GLOBALCONSTANTS DefaultPool_PI_Numeric (* Numeric object pool constants (ID, Scale, Offset, Decimals) *)
  PACKAGE Uebungen::const::UT::PI;
  VAR_GLOBAL CONSTANT
    OutputNumber_c1_N : logiBUS::utils::conversion::phys::NumericObjectPool_S := (u16ObjId := 12001, r32Scale := 1.0, i32Offset := 0, u8Decimals := 0);
    OutputNumber_c9_N : logiBUS::utils::conversion::phys::NumericObjectPool_S := (u16ObjId := 12009, r32Scale := 1.0, i32Offset := 0, u8Decimals := 0);
    OutputNumber_c10_N : logiBUS::utils::conversion::phys::NumericObjectPool_S := (u16ObjId := 12010, r32Scale := 1.0, i32Offset := 0, u8Decimals := 0);
    OutputNumber_c11_N : logiBUS::utils::conversion::phys::NumericObjectPool_S := (u16ObjId := 12011, r32Scale := 1.0, i32Offset := 0, u8Decimals := 0);
    OutputNumber_c12_N : logiBUS::utils::conversion::phys::NumericObjectPool_S := (u16ObjId := 12012, r32Scale := 1.0, i32Offset := 0, u8Decimals := 0);
    OutputNumber_c2_N : logiBUS::utils::conversion::phys::NumericObjectPool_S := (u16ObjId := 12013, r32Scale := 1.0, i32Offset := 0, u8Decimals := 0);
    OutputNumber_c3_N : logiBUS::utils::conversion::phys::NumericObjectPool_S := (u16ObjId := 12014, r32Scale := 1.0, i32Offset := 0, u8Decimals := 0);
    OutputNumber_c4_N : logiBUS::utils::conversion::phys::NumericObjectPool_S := (u16ObjId := 12015, r32Scale := 1.0, i32Offset := 0, u8Decimals := 0);
    OutputNumber_c5_N : logiBUS::utils::conversion::phys::NumericObjectPool_S := (u16ObjId := 12016, r32Scale := 1.0, i32Offset := 0, u8Decimals := 0);
    OutputNumber_c6_N : logiBUS::utils::conversion::phys::NumericObjectPool_S := (u16ObjId := 12017, r32Scale := 1.0, i32Offset := 0, u8Decimals := 0);
    OutputNumber_c7_N : logiBUS::utils::conversion::phys::NumericObjectPool_S := (u16ObjId := 12018, r32Scale := 1.0, i32Offset := 0, u8Decimals := 0);
    OutputNumber_c8_N : logiBUS::utils::conversion::phys::NumericObjectPool_S := (u16ObjId := 12019, r32Scale := 1.0, i32Offset := 0, u8Decimals := 0);
    OutputNumber_Tick_N : logiBUS::utils::conversion::phys::NumericObjectPool_S := (u16ObjId := 12020, r32Scale := 1.0, i32Offset := 0, u8Decimals := 0);
    OutputNumber_PI_I01_FREQ_N : logiBUS::utils::conversion::phys::NumericObjectPool_S := (u16ObjId := 12021, r32Scale := 1.0, i32Offset := 0, u8Decimals := 0);
    OutputNumber_PI_I01_COUNT_N : logiBUS::utils::conversion::phys::NumericObjectPool_S := (u16ObjId := 12022, r32Scale := 1.0, i32Offset := 0, u8Decimals := 0);
    OutputNumber_PI_I02_FREQ_N : logiBUS::utils::conversion::phys::NumericObjectPool_S := (u16ObjId := 12023, r32Scale := 1.0, i32Offset := 0, u8Decimals := 0);
    OutputNumber_PI_I02_COUNT_N : logiBUS::utils::conversion::phys::NumericObjectPool_S := (u16ObjId := 12024, r32Scale := 1.0, i32Offset := 0, u8Decimals := 0);
    OutputNumber_PI_I03_FREQ_N : logiBUS::utils::conversion::phys::NumericObjectPool_S := (u16ObjId := 12025, r32Scale := 1.0, i32Offset := 0, u8Decimals := 0);
    OutputNumber_PI_I03_COUNT_N : logiBUS::utils::conversion::phys::NumericObjectPool_S := (u16ObjId := 12026, r32Scale := 1.0, i32Offset := 0, u8Decimals := 0);
    OutputNumber_PI_I04_FREQ_N : logiBUS::utils::conversion::phys::NumericObjectPool_S := (u16ObjId := 12027, r32Scale := 1.0, i32Offset := 0, u8Decimals := 0);
    OutputNumber_PI_I04_COUNT_N : logiBUS::utils::conversion::phys::NumericObjectPool_S := (u16ObjId := 12028, r32Scale := 1.0, i32Offset := 0, u8Decimals := 0);
    OutputNumber_PI_I05_FREQ_N : logiBUS::utils::conversion::phys::NumericObjectPool_S := (u16ObjId := 12029, r32Scale := 1.0, i32Offset := 0, u8Decimals := 0);
    OutputNumber_PI_I05_COUNT_N : logiBUS::utils::conversion::phys::NumericObjectPool_S := (u16ObjId := 12030, r32Scale := 1.0, i32Offset := 0, u8Decimals := 0);
    OutputNumber_PI_I06_FREQ_N : logiBUS::utils::conversion::phys::NumericObjectPool_S := (u16ObjId := 12031, r32Scale := 1.0, i32Offset := 0, u8Decimals := 0);
    OutputNumber_PI_I06_COUNT_N : logiBUS::utils::conversion::phys::NumericObjectPool_S := (u16ObjId := 12032, r32Scale := 1.0, i32Offset := 0, u8Decimals := 0);
    OutputNumber_PI_I07_FREQ_N : logiBUS::utils::conversion::phys::NumericObjectPool_S := (u16ObjId := 12033, r32Scale := 1.0, i32Offset := 0, u8Decimals := 0);
    OutputNumber_PI_I07_COUNT_N : logiBUS::utils::conversion::phys::NumericObjectPool_S := (u16ObjId := 12034, r32Scale := 1.0, i32Offset := 0, u8Decimals := 0);
    OutputNumber_PI_I08_FREQ_N : logiBUS::utils::conversion::phys::NumericObjectPool_S := (u16ObjId := 12035, r32Scale := 1.0, i32Offset := 0, u8Decimals := 0);
    OutputNumber_PI_I08_COUNT_N : logiBUS::utils::conversion::phys::NumericObjectPool_S := (u16ObjId := 12036, r32Scale := 1.0, i32Offset := 0, u8Decimals := 0);
    NumberVariable_PI_FREQ_I01_N : logiBUS::utils::conversion::phys::NumericObjectPool_S := (u16ObjId := 21000, r32Scale := 1.0, i32Offset := 0, u8Decimals := 0);
    NumberVariable_PI_FREQ_I02_N : logiBUS::utils::conversion::phys::NumericObjectPool_S := (u16ObjId := 21001, r32Scale := 1.0, i32Offset := 0, u8Decimals := 0);
    NumberVariable_PI_FREQ_I03_N : logiBUS::utils::conversion::phys::NumericObjectPool_S := (u16ObjId := 21002, r32Scale := 1.0, i32Offset := 0, u8Decimals := 0);
    NumberVariable_PI_FREQ_I04_N : logiBUS::utils::conversion::phys::NumericObjectPool_S := (u16ObjId := 21003, r32Scale := 1.0, i32Offset := 0, u8Decimals := 0);
    NumberVariable_PI_FREQ_I05_N : logiBUS::utils::conversion::phys::NumericObjectPool_S := (u16ObjId := 21004, r32Scale := 1.0, i32Offset := 0, u8Decimals := 0);
    NumberVariable_PI_FREQ_I06_N : logiBUS::utils::conversion::phys::NumericObjectPool_S := (u16ObjId := 21005, r32Scale := 1.0, i32Offset := 0, u8Decimals := 0);
    NumberVariable_PI_FREQ_I07_N : logiBUS::utils::conversion::phys::NumericObjectPool_S := (u16ObjId := 21006, r32Scale := 1.0, i32Offset := 0, u8Decimals := 0);
    NumberVariable_PI_FREQ_I08_N : logiBUS::utils::conversion::phys::NumericObjectPool_S := (u16ObjId := 21007, r32Scale := 1.0, i32Offset := 0, u8Decimals := 0);
    NumberVariable_PI_COUNT_I01_N : logiBUS::utils::conversion::phys::NumericObjectPool_S := (u16ObjId := 21008, r32Scale := 1.0, i32Offset := 0, u8Decimals := 0);
    NumberVariable_PI_COUNT_I02_N : logiBUS::utils::conversion::phys::NumericObjectPool_S := (u16ObjId := 21009, r32Scale := 1.0, i32Offset := 0, u8Decimals := 0);
    NumberVariable_PI_COUNT_I03_N : logiBUS::utils::conversion::phys::NumericObjectPool_S := (u16ObjId := 21010, r32Scale := 1.0, i32Offset := 0, u8Decimals := 0);
    NumberVariable_PI_COUNT_I04_N : logiBUS::utils::conversion::phys::NumericObjectPool_S := (u16ObjId := 21011, r32Scale := 1.0, i32Offset := 0, u8Decimals := 0);
    NumberVariable_PI_COUNT_I05_N : logiBUS::utils::conversion::phys::NumericObjectPool_S := (u16ObjId := 21012, r32Scale := 1.0, i32Offset := 0, u8Decimals := 0);
    NumberVariable_PI_COUNT_I06_N : logiBUS::utils::conversion::phys::NumericObjectPool_S := (u16ObjId := 21013, r32Scale := 1.0, i32Offset := 0, u8Decimals := 0);
    NumberVariable_PI_COUNT_I07_N : logiBUS::utils::conversion::phys::NumericObjectPool_S := (u16ObjId := 21014, r32Scale := 1.0, i32Offset := 0, u8Decimals := 0);
    NumberVariable_PI_COUNT_I08_N : logiBUS::utils::conversion::phys::NumericObjectPool_S := (u16ObjId := 21015, r32Scale := 1.0, i32Offset := 0, u8Decimals := 0);
  END_VAR
END_GLOBALCONSTANTS
